// TIA Portal V20 export
DATA_BLOCK "BK14"   // DB258
// stored: MemoryReserve 100
   VAR
      "X10-1 HIPOT TAB CONTACTOR BACKWARD" : Bool;
      "X11-1 HIPOT TAB CONTACTOR LEFT OPEN" : Bool;
      "X12-1 HIPOT TAB CONTACTOR RIGHT OPEN" : Bool;
      "X13-1 SPARE" : Bool;
      "X14-1 SPARE" : Bool;
      "X15-1 HIPOT&THICKNESS STAGE LIFT FRONT DOWN" : Bool;
      "X16-1 HIPOT&THICKNESS STAGE LIFT REAR DOWN" : Bool;
      "X17-1 SPARE" : Bool;
      "X10-2 HIPOT TAB CONTACTOR FORWARD" : Bool;
      "X11-2 HIPOT TAB CONTACTOR LEFT CLOSE" : Bool;
      "X12-2 HIPOT TAB CONTACTOR RIGHT CLOSE" : Bool;
      "X13-2 SPARE" : Bool;
      "X14-2 SPARE" : Bool;
      "X15-2 INSPECTION STAGE LIFT FRONT UP" : Bool;
      "X16-2 INSPECTION STAGE LIFT REAR UP" : Bool;
      "X17-2 SPARE" : Bool;
   END_VAR
BEGIN
END_DATA_BLOCK
